// TIA Portal V20 export
TYPE "typeEstopZoneSummary"
// stored: Access Published, IsFailsafeCompliant true, Namespace Safety
   STRUCT
      insideEstopOk : Bool;
      outsideEstopOk : Bool;
      allEstopOk : Bool;
   END_STRUCT;
END_TYPE
